(* CODESYS project FU_wBitGet.xml

Project tree, tasks and I/O mapping:
  function FU_wBitGet [ST]
*)

// FU_wBitGet
//This function get the bit value from a variable
// |**Version**|**Author**| **Date** |**Changes**
// | 1         | NSN      | 11-01-19 | Creation
FUNCTION FU_wBitGet : BOOL
VAR_INPUT
	wVar	:WORD;		//The value to work with
	bIndex	:BYTE;		//Which bit to get	
END_VAR

FU_wBitGet		:=		(wVar AND SHL(1,bIndex)) <> 0;

END_FUNCTION
